// TIA Portal V17 export
// export: Created 2025-06-26T06:49:30.9421717Z, ExportSetting WithDefaults, DisplayName Totally Integrated Automation Portal, DisplayVersion V17 Update 8, DisplayName TIA Portal Openness, DisplayVersion V17 Update 8, DisplayName TIA Portal Version Control Interface, DisplayVersion V17, DisplayName STEP 7 Professional, DisplayVersion V17 Update 8, DisplayName STEP 7 Safety, DisplayVersion V17 Update 6, DisplayName WinCC Advanced, DisplayVersion V17 Update 8
TYPE "stPinchControl"
// stored: IsFailsafeCompliant false
   STRUCT
      bEnable : Bool;   // 1 = enable from HMI, 0 = disable from HMI
      bFault : Bool;   // 1 = fault, 0 = ok
      nMode : USInt;   // 0 = offline, 1 = auto, 2 = manual
      fSetpoint : Real;   // Selected setpoint
      fPV : Real;   // Process value
      Regulator : "stPID_Regulator";
   END_STRUCT;
END_TYPE
